{attribute addProperty BoxType "EJ9505-0000-0016"}
{attribute addProperty Id "Power_OKAT %I*BOOL811OverloadAT %I*BOOL812"}
{attribute addProperty CRC "3527607142"}
{attribute addProperty SizeInBites "16"}
{attribute addProperty SizeInBytes "2"}
TYPE Status_Uo_D2430366 :
STRUCT
	{attribute addProperty Name "Power_OK"}
	Power_OK AT %I* : BOOL;
	{attribute addProperty Name "Overload"}
	Overload AT %I* : BOOL;
END_STRUCT
END_TYPE

(* stored: Version 1.2.0.0, ProductVersion 3.1.4024.9
   DUT Status_Uo_D2430366: Id {62218b68-5a7c-4f26-b242-1614190f2e2c} *)
